// minimal Unit for the base suite: 2-step looping chain, one wait-classed step
FUNCTION_BLOCK FB_ProbeUnit EXTENDS FB_UnitBase
VAR_INPUT
    SimA, SimB : BOOL;
    SimFault : BOOL;                    // deterministic fault injection for base-path tests
END_VAR
VAR_OUTPUT
    ModeChangedCount : UDINT;
    ModeExitCount : UDINT;
    ModeExitFirstCount : UDINT;
    LastNewMode : E_Mode;
    LastOldMode : E_Mode;
    LastRequestedMode : E_Mode;
END_VAR

Cyclic();

METHOD Setup : BOOL
VAR_INPUT
    Name : STRING(80);
END_VAR
_M_SetName(Name);
StallTime := T#0S;                       // test: stall pending fires immediately
Setup := TRUE;
END_METHOD

METHOD PROTECTED _M_Dispatch
CASE _step OF
    10:
        _M_SetStep(StepNo := 100, StepName := 'project.test.stepA', Awaits := 0,
            AwaitingLabel := '', Class := E_TimeClass.WORK, ExpectedTime := T#0S);
        IF SimFault THEN
            _M_Fault(E_Reason.TEST_FAULT, 'forced Unit fault');
        ELSIF SimA THEN
            _step := 20;
        END_IF
    20:
        _M_SetStep(StepNo := 200, StepName := 'project.test.stepB', Awaits := 0,
            AwaitingLabel := '', Class := E_TimeClass.WAIT_UPSTREAM, ExpectedTime := T#0S);
        IF SimB THEN
            _step := 30;
        END_IF
    30:
        IF _M_EndOfCycle() THEN
            _step := 10;
        END_IF
ELSE
    _M_Fault(E_Reason.STEP_STALLED, 'undefined step');
END_CASE
END_METHOD

METHOD PROTECTED OnModeChanged : DINT
VAR_INPUT
    NewMode : E_Mode;
    OldMode : E_Mode;
END_VAR
OnModeChanged := SUPER^.OnModeChanged(
    NewMode := NewMode, OldMode := OldMode);
ModeChangedCount := ModeChangedCount + 1;
LastNewMode := NewMode;
LastOldMode := OldMode;
END_METHOD

METHOD PROTECTED OnModeExit : DINT
VAR_INPUT
    FirstCall : BOOL;
    RequestedMode : E_Mode;
END_VAR
// This probe wants the default immediate cancel, so the base call is intentional.
OnModeExit := SUPER^.OnModeExit(
    FirstCall := FirstCall, RequestedMode := RequestedMode);
ModeExitCount := ModeExitCount + 1;
IF FirstCall THEN
    ModeExitFirstCount := ModeExitFirstCount + 1;
END_IF
LastRequestedMode := RequestedMode;
END_METHOD

END_FUNCTION_BLOCK

(* stored: Version 1.1.0.1, ProductVersion 3.1.4024.12
   POU FB_ProbeUnit: Id {a1676a86-f95f-460f-93ca-ed94ca5c7c5d}, SpecialFunc None
   Method Setup: Id {5b7a8b1b-03fd-4d4e-b0d2-5821d68d823c}
   Method _M_Dispatch: Id {2d5f574b-01d6-4291-a6ce-b24e805a7176}
   Method OnModeChanged: Id {c8d47169-ae9c-42b2-a7bc-8b4fbc0bab15}
   Method OnModeExit: Id {1c73f57f-9a1f-43d6-a9a0-2fe455382bca} *)
